// Mitsubishi GX Works2 project: LRI - PLC - SEMAFARO ST   PLC: Q03UDV

// task Task_01 (event TRUE, interval 0, priority 31): POU_01

PROGRAM POU_01
VAR
  stSemafaro_1 : stSemafaro;
END_VAR
stSemafaro_1(i_Habilitar:= 1 ,i_Tempo_Verde_Ligado:= 5 ,i_Tempo_Amarelo_Ligado:= 5 ,t_tempo_Vermelho_Vermelho:= 4 ,i_Quantidade_Pisca_Verde:= 4 ,
	i_Quantidade_Pisca_Amarelo:= 4 ,i_Quantidade_Pisca_Vermelho:=4 );
END_PROGRAM

FUNCTION_BLOCK stSemafaro
VAR_INPUT
  i_Habilitar : BOOL;
  i_Tempo_Verde_Ligado : INT;
  i_Tempo_Amarelo_Ligado : INT;
  t_tempo_Vermelho_Vermelho : INT;
  i_Quantidade_Pisca_Verde : INT;
  i_Quantidade_Pisca_Amarelo : INT;
  i_Quantidade_Pisca_Vermelho : INT;
END_VAR
VAR
  x_Contadador_Pisca : ARRAY [0..5] OF INT;
  rtTrigger : R_TRIG;
  x_Contador_Estado : ARRAY [0..4] OF INT;
  t_Tempo_Atual : INT;
END_VAR
VAR_OUTPUT
  stg_Estados_Semafaro : ARRAY [0..5] OF INT;
END_VAR
(*Verificar se o semafaro está habilitado*)
IF i_Habilitar = TRUE THEN
	
	(*Verificar se o tempo do sinal verde do semafaro 1 é menor que o tempo atual*)
	IF i_Tempo_Verde_Ligado >= t_Tempo_Atual THEN
	  	stg_Estados_Semafaro[0]:= 1;
		stg_Estados_Semafaro[1] := 0; 
		stg_Estados_Semafaro[2] := 0; 
		stg_Estados_Semafaro[3] := 0; 
		stg_Estados_Semafaro[4] := 0; 
		stg_Estados_Semafaro[5] := 1; 
		
	(*Condição para sinal verde do semafaro 1 piscar*)	
	ELSIF i_Quantidade_Pisca_Verde >=  x_Contadador_Pisca[0] THEN
		
						rtTrigger(_CLK:=SM412);
						IF rtTrigger.Q THEN
						stg_Estados_Semafaro[0] := 0;
						x_Contadador_Pisca[0] := x_Contadador_Pisca[0]+1;
						ELSE
						stg_Estados_Semafaro[0]:= 1;
						END_IF;
			(*contador auxiliar para somar o tempo atual mais o tempo que o amarelo deve ficar ligado*)	
			x_Contador_Estado[0] := t_Tempo_Atual + i_Tempo_Amarelo_Ligado;
	
	(*Verificar se o tempo do sinal amarelo do semafaro 1 é menor que o tempo atual*)	
	ELSIF x_Contador_Estado[0] >= t_Tempo_Atual THEN	
	 	stg_Estados_Semafaro[0] := 0; 
		stg_Estados_Semafaro[1] := 1; 
		stg_Estados_Semafaro[2] := 0; 
		stg_Estados_Semafaro[3] := 0; 
		stg_Estados_Semafaro[4] := 0; 
		stg_Estados_Semafaro[5] := 1;
		
	(*Condição para sinal amarelo do semafaro 1 piscar*)
	ELSIF i_Quantidade_Pisca_Amarelo >=  x_Contadador_Pisca[1] THEN
		
						rtTrigger(_CLK:=SM412);
						IF rtTrigger.Q THEN
						stg_Estados_Semafaro[1] := 0;
						x_Contadador_Pisca[1] := x_Contadador_Pisca[1]+1;				
						ELSE
						stg_Estados_Semafaro[1]:= 1;
						END_IF;			
		(*contador auxiliar para somar o tempo atual mais o tempo que o vermelho deve ficar ligado*)
		x_Contador_Estado[1] := t_Tempo_Atual + t_tempo_Vermelho_Vermelho;
	
	(*Verificar se o tempo do sinal vermelho do semafaro 1 é menor que o tempo atual*)	
	ELSIF x_Contador_Estado[1] >= t_Tempo_Atual THEN
		stg_Estados_Semafaro[0] := 0; 
		stg_Estados_Semafaro[1] := 0; 
		stg_Estados_Semafaro[2] := 1; 
		stg_Estados_Semafaro[3] := 0; 
		stg_Estados_Semafaro[4] := 0; 
		stg_Estados_Semafaro[5] := 1;
		
	(*Condição para sinal vermelho do semafaro 1 piscar*)
	ELSIF i_Quantidade_Pisca_Vermelho >=  x_Contadador_Pisca[2] THEN
		
						rtTrigger(_CLK:=SM412);
						IF rtTrigger.Q THEN
						stg_Estados_Semafaro[2] := 0;
						x_Contadador_Pisca[2] := x_Contadador_Pisca[2]+1;
						ELSE
						stg_Estados_Semafaro[2]:= 1;
						END_IF;		
		(*contador auxiliar para somar o tempo atual mais o tempo que o verde deve ficar ligado*)				
		x_Contador_Estado[2] := t_Tempo_Atual + i_Tempo_Verde_Ligado;
	
	(*Verificar se o tempo do sinal verde do semafaro 2 é menor que o tempo atual*)	
	ELSIF x_Contador_Estado[2] >= t_Tempo_Atual THEN	
		stg_Estados_Semafaro[0] := 0; 
		stg_Estados_Semafaro[1] := 0; 
		stg_Estados_Semafaro[2] := 1; 
		stg_Estados_Semafaro[3] := 1; 
		stg_Estados_Semafaro[4] := 0; 
		stg_Estados_Semafaro[5] := 0;
		
	(*Condição para sinal verde do semafaro 2 piscar*)
	ELSIF i_Quantidade_Pisca_Verde >=  x_Contadador_Pisca[3] THEN
		 
						rtTrigger(_CLK:=SM412);
						IF rtTrigger.Q THEN
						stg_Estados_Semafaro[3] := 0;
						x_Contadador_Pisca[3] := x_Contadador_Pisca[3]+1;
						ELSE
						stg_Estados_Semafaro[3]:= 1;
						END_IF;	
		(*contador auxiliar para somar o tempo atual mais o tempo que o amarelo deve ficar ligado*)						
		x_Contador_Estado[3] := t_Tempo_Atual + i_Tempo_Amarelo_Ligado;
	
	(*Verificar se o tempo do sinal amarelo do semafaro 2 é menor que o tempo atual*)	
	ELSIF x_Contador_Estado[3] >= t_Tempo_Atual THEN	
		stg_Estados_Semafaro[0] := 0; 
		stg_Estados_Semafaro[1] := 0; 
		stg_Estados_Semafaro[2] := 1; 
		stg_Estados_Semafaro[3] := 0; 
		stg_Estados_Semafaro[4] := 1; 
		stg_Estados_Semafaro[5] := 0;
	
	(*Condição para sinal amarelo do semafaro 2 piscar*)
	ELSIF i_Quantidade_Pisca_Amarelo >=  x_Contadador_Pisca[4] THEN
		 
						rtTrigger(_CLK:=SM412);
						IF rtTrigger.Q THEN
						stg_Estados_Semafaro[4] := 0;
						x_Contadador_Pisca[4] := x_Contadador_Pisca[4]+1;
						ELSE
						stg_Estados_Semafaro[4]:= 1;
						END_IF;	
		(*contador auxiliar para somar o tempo atual mais o tempo que o vermelho deve ficar ligado*)					
		x_Contador_Estado[4] := t_Tempo_Atual + t_tempo_Vermelho_Vermelho;
	
	(*Verificar se o tempo do sinal vermelho do semafaro 2 é menor que o tempo atual*)	
	ELSIF  x_Contador_Estado[4]  >=  t_Tempo_Atual THEN	
		stg_Estados_Semafaro[0] := 0; 
		stg_Estados_Semafaro[1] := 0; 
		stg_Estados_Semafaro[2] := 1; 
		stg_Estados_Semafaro[3] := 0; 
		stg_Estados_Semafaro[4] := 0; 
		stg_Estados_Semafaro[5] := 1;
	
	(*Condição para sinal vermelho do semafaro 2 piscar*)	
	ELSIF i_Quantidade_Pisca_Vermelho >=  x_Contadador_Pisca[5] THEN
		 
						rtTrigger(_CLK:=SM412);
						IF rtTrigger.Q THEN
						stg_Estados_Semafaro[5] := 0;
						x_Contadador_Pisca[5] := x_Contadador_Pisca[5]+1;
						ELSE
						stg_Estados_Semafaro[5]:= 1;
						END_IF;	
						
	(*Resetar variaveis temporais para reiniciar tudo*)					
	ELSE 	
		t_Tempo_Atual := 0 ;
		x_Contador_Estado[0] := 0; 
		x_Contador_Estado[1] := 0; 
		x_Contador_Estado[2] := 0; 
		x_Contador_Estado[3] := 0; 
		x_Contador_Estado[4] := 0; 	
		x_Contadador_Pisca[0] := 0;
		x_Contadador_Pisca[1] := 0;
		x_Contadador_Pisca[2] := 0;
		x_Contadador_Pisca[3] := 0;
		x_Contadador_Pisca[4] := 0;
		x_Contadador_Pisca[5] := 0;
	END_IF;	
	
		(*Contador baseado no SM412 que gera um pulso a cada um segundo*)
		rtTrigger(_CLK:=SM412);
			IF rtTrigger.Q THEN
				t_Tempo_Atual:= t_Tempo_Atual+1;
			END_IF;
	
END_IF	;
END_FUNCTION_BLOCK
